FUNCTION_BLOCK FT_PT1_AR (* AR-Adapter-Wrapper um OSCAT FT_PT1 (PT1-Tiefpassfilter) - bruckt zwischen adapter und OSCAT, ohne dass eine der beiden Basisbibliotheken von der anderen abhaengt. TM (Zeitkonstante) als ATM-Socket (kein Klartext-InputVar, sauber initialisierbar ueber initval_ATM), K als Klartext-InputVar durchgereicht (Default 1.0) *)
  (* Standard: 61499-2; Description: Copyright (c) 2026 Meisterschulen am Ostbahnhof This program and the accompanying materials are made available under the terms of the Eclipse Public License 2.0 which is available at https://www.eclipse.org/legal/epl-2.0/ SPDX-License-Identifier: EPL-2.0 *)
  (* Version 1.3, 2026-09-26, Franz Höpfinger, Meisterschulen am Ostbahnhof, Schema-Fix: Sockets/Plugs-Reihenfolge im InterfaceList vertauscht (IDE-Resave hatte Plugs vor Sockets geschrieben) - block-common.xsd verlangt strikt Sockets vor Plugs, sonst schlaegt validate.py mit 'Element Sockets: This element is not expected' fehl. Beim Gegenchecken des Review-Bot-Funds zu FT_PT1 v1.2 (fehlendes Organization-Attribut) entdeckt, unabhaengiges Problem. *)
  (* Version 1.2, 2026-09-26, Franz Höpfinger, Meisterschulen am Ostbahnhof, Franz: 'Sind alle WITH dafuer noch passend?' - Kommentare/Doku zu RST korrigiert, beschrieben bisher noch das alte Verhalten (out := K * in direkt in RST). Seit FT_PT1 v1.3 (Review-Bot-Fund auf training1 PR #269) setzt RST nur noch init:=FALSE, das Seeding passiert im naechsten REQ mit frisch abgetastetem in. With-Var-Deklarationen selbst unveraendert/weiterhin korrekt (REQ braucht in/TM/K, RST brauchte und braucht keine - referenziert weder in noch TM noch K); CNF (delta_t/out) bleibt syntaktisch gueltig, traegt beim RST-Fall aber jetzt bewusst die unveraenderten alten Werte (kein Bug, siehe Doku unten). *)
  (* Version 1.1, 2026-09-17, Franz Höpfinger, Meisterschulen am Ostbahnhof, Franz: 'RST muss raus gefuehrt werden' - neues EventInput RST, 1:1 durchgereicht an FT_PT1.RST (analog INIT/EINIT), seit FT_PT1.fbt v1.1 das RST-Event wieder hat. Kein zusaetzlicher CNF-Pfad noetig: FT_PT1.CNF (RST und REQ feuern beide denselben CNF-Ausgang) ist bereits an E_D_FF_ANY.CLK angeschlossen. Franz: 'K muss ein WITH Konstrukt haben, z.B. mit INIT' - K jetzt als With-Var am INIT-Event deklariert (analog QI/PARAMS bei den IXA/IX-Bausteinen), statt nur ueber eine formlose durchgehende DataConnection - K ist ein statischer Konfigurationswert, kein pro-Zyklus-Datum wie in/out. *)
  (* Version 1.0, 2026-09-17, Franz Höpfinger, Meisterschulen am Ostbahnhof, Initial implementation of FT_PT1_AR wrapper FB (Franz: 'portiere diese Bausteine hier her', OSCAT_basic FT_PT1.TcPOU) - E_D_FF_ANY als Aenderungsfilter (EO/AR_OUT.E1 nur bei tatsaechlicher Wertaenderung), analog ROUND_AR/FT_DERIV_AR in diesem Projekt. TM als ATM-Socket statt Klartext-InputVar (Section 13 des iec61499-creator-Skills: TIME-Konfigurationswerte gehoeren auf einen Adapter-Socket, initialisiert per initval_ATM an der Instanziierungsstelle - gleiches Muster wie AE_DELAY/ASR2_DELAY). *)
  PACKAGE OSCAT_adapter::Control;
  (* Documentation:
  FT_PT1_AR
   🇩🇪 Deutsch
   AR-Adapter-Wrapper um OSCAT::Basic::POUs::Engineering::Control::FT_PT1 (PT1-Tiefpassfilter mit programmierbarer Zeitkonstante TM und Faktor K). TM ist ein ATM-Socket (kein Klartext-InputVar) - an der Instanziierungsstelle ueber adapter::types::unidirectional::TIME::initval::initval_ATM zu initialisieren, damit die Zeitkonstante sauber ueber INIT/INITO gesetzt wird (Section 13 des iec61499-creator-Skills: TIME-Konfigurationswerte gehoeren nicht auf einen nackten InputVar). K (Faktor, Default 1.0) bleibt ein Klartext-InputVar, ist aber als With-Var am INIT-Event deklariert (statt nur formlos durchgehend verdrahtet) - ein statischer Konfigurationswert wie bei den IXA/IX-Bausteinen (QI/PARAMS als With-Var an INIT), nicht wie in/out ein pro-Zyklus-Datum.
   Reine Adapter-Grenze
    - AR_IN (Socket, AR): Eingangssignal (REAL)
   - TM (Socket, ATM): Zeitkonstante
   - AR_OUT (Plug, AR): gefilterter Ausgangswert (REAL)
    E_D_FF_ANY filtert Aenderungen: AR_OUT.E1 feuert nur, wenn sich der gefilterte Wert seit dem letzten Aufruf tatsaechlich geaendert hat - gleiches Muster wie bei ROUND_AR/FT_DERIV_AR in diesem Projekt.
   INIT/INITO werden 1:1 an FT_PT1.EINIT/.INITO durchgereicht - wie bei den uebrigen Service-Wrappern in diesem Repo. Bleibt INIT unverdrahtet, feuert es einmalig beim Deployment automatisch (Standardkonvention fuer unverdrahtete EInit-Events).
   RST (EventInput) wird 1:1 an FT_PT1.RST durchgereicht - invalidiert nur den Zustand (init:=FALSE), ohne selbst out zu setzen: RST hat kein in-With-Var und koennte sonst mit einem veralteten oder (bei TM.E1-getriggertem RST vor der ersten Messung) noch nie gesetzten Wert falsch seeden. Das naechste REQ (mit garantiert frischem in per With-Var) macht das eigentliche Seeding (out := K * in) selbst inline (FT_PT1 v1.3). Kein eigener CNF-Pfad noetig: FT_PT1.CNF feuert bei RST genauso wie bei REQ und ist bereits an E_D_FF_ANY.CLK angeschlossen - traegt beim RST-Fall allerdings noch die alten delta_t/out-Werte (unveraendert seit dem letzten REQ), AR_OUT.E1 feuert also erst wieder beim naechsten REQ, sobald sich der Wert dadurch tatsaechlich aendert.
   Warum ein eigener Wrapper?
   FT_PT1 ist ein reines OSCAT-FB (SimpleFB, zustandsbehaftet: last/tx/init) ohne Adapter-Schnittstelle. adapter soll nicht von OSCAT abhaengen (und umgekehrt) - die Bruecke liegt daher in diesem dritten Bibliotheksprojekt (OSCAT_adapter), das von beiden abhaengt.
   🇬🇧 English
   AR-adapter wrapper around OSCAT::Basic::POUs::Engineering::Control::FT_PT1 (PT1 low-pass filter with programmable time constant TM and factor K). TM is an ATM socket (not a plain InputVar) - initialize it at the instantiation site via adapter::types::unidirectional::TIME::initval::initval_ATM so the time constant is set cleanly via INIT/INITO (per section 13 of the iec61499-creator skill: TIME configuration values do not belong on a bare InputVar). K (factor, default 1.0) stays a plain InputVar, but is declared as a With-Var on the INIT event (instead of just an informally always-wired connection) - a static configuration value like QI/PARAMS on the IXA/IX blocks (With-Var on INIT), not a per-cycle datum like in/out.
   Pure adapter boundary
    - AR_IN (socket, AR): input signal (REAL)
   - TM (socket, ATM): time constant
   - AR_OUT (plug, AR): filtered output value (REAL)
    E_D_FF_ANY filters changes: AR_OUT.E1 only fires when the filtered value actually changed since the last call - same pattern as ROUND_AR/FT_DERIV_AR in this project.
   INIT/INITO are passed through 1:1 to FT_PT1.EINIT/.INITO - as with the other service wrappers in this repo. If INIT is left unconnected, it auto-fires once at deployment (standard convention for unconnected EInit events).
   RST (event input) is passed through 1:1 to FT_PT1.RST - only invalidates the state (init:=FALSE) without setting out itself: RST has no in With-Var and could otherwise seed with a stale or (when triggered via TM.E1 before the first measurement) never-set value. The next REQ (with guaranteed-fresh in via its own With-Var) does the actual seeding (out := K * in) inline (FT_PT1 v1.3). No separate CNF path needed: FT_PT1.CNF fires on RST just like on REQ and is already wired to E_D_FF_ANY.CLK - though on the RST path it still carries the old, unchanged delta_t/out values, so AR_OUT.E1 only fires again on the next REQ once the value actually changes.
   Why a dedicated wrapper?
   FT_PT1 is a plain OSCAT FB (SimpleFB, stateful: last/tx/init) with no adapter interface. adapter must not depend on OSCAT (nor vice versa) - the bridge lives in this third library project (OSCAT_adapter), which depends on both.
  *)
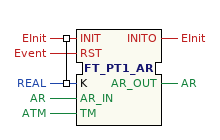
  EVENT_INPUT
    INIT : EInit WITH K; (* Service Initialization (durchgereicht an FT_PT1.EINIT) *)
    RST; (* Filter zuruecksetzen (durchgereicht an FT_PT1.RST) - invalidiert nur den Zustand (init:=FALSE), das naechste REQ seedet mit frisch abgetastetem in (FT_PT1 v1.3) *)
  END_EVENT
  EVENT_OUTPUT
    INITO : EInit; (* Initialization Confirm *)
  END_EVENT
  VAR_INPUT
    K : REAL := 1.0; (* Faktor (durchgereicht an FT_PT1.K) *)
  END_VAR
  SOCKETS
    AR_IN : adapter::types::unidirectional::AR; (* Eingangssignal (REAL) *)
    TM : adapter::types::unidirectional::ATM; (* Zeitkonstante (durchgereicht an FT_PT1.TM) *)
  END_SOCKETS
  PLUGS
    AR_OUT : adapter::types::unidirectional::AR; (* Gefilterter Ausgangswert (REAL, durchgereicht von FT_PT1.out) *)
  END_PLUGS
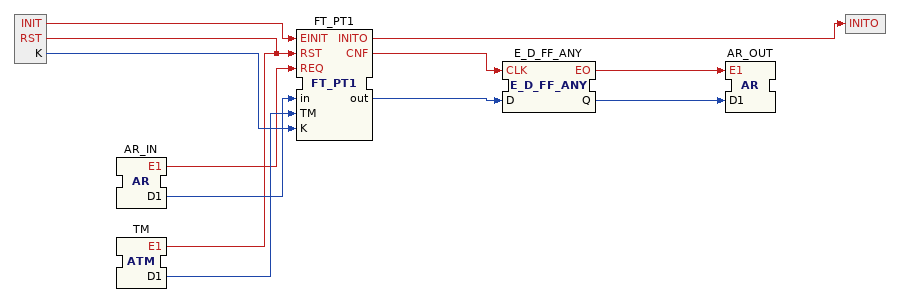
  FBS
    FT_PT1 : OSCAT::Basic::POUs::Engineering::Control::FT_PT1;
    E_D_FF_ANY : iec61499::events::E_D_FF_ANY;
  END_FBS
  EVENT_CONNECTIONS
    INIT TO FT_PT1.EINIT;
    FT_PT1.INITO TO INITO;
    RST TO FT_PT1.RST;
    AR_IN.E1 TO FT_PT1.REQ;
    FT_PT1.CNF TO E_D_FF_ANY.CLK;
    E_D_FF_ANY.EO TO AR_OUT.E1;
    TM.E1 TO FT_PT1.RST;
  END_CONNECTIONS
  DATA_CONNECTIONS
    AR_IN.D1 TO FT_PT1.in;
    TM.D1 TO FT_PT1.TM;
    K TO FT_PT1.K;
    FT_PT1.out TO E_D_FF_ANY.D;
    E_D_FF_ANY.Q TO AR_OUT.D1;
  END_CONNECTIONS
END_FUNCTION_BLOCK
